// TIA Portal project "9input_to_4output" (V14)

(* hardware
DEVICE "S7-1200 station_1"  S7-1200 Station
   slot 0: "Rack_0"  S7-1200 Rack  Rack  V1.0
   slot 1: "PLC_1"  CPU 1214C DC/DC/DC  6ES7 214-1AG40-0XB0  V4.2
DEVICE "HMI_1"  KTP700 Basic PN
   slot 0: "KTP700 Basic PN"  KTP700 Basic PN  6AV2 123-2GB03-0AX0  14.0.1.0
   slot 1: "HMI_RT_1"  KTP700 Basic PN  6AV2 123-2GB03-0AX0  14.0.1.0
   slot 5: "HMI_1.IE_CP_1"  PROFINET Interface  14.0.1.0
      slot 1: "PROFINET Interface_1"  PROFINET Interface
         slot 1: "Port_1"  Port
*)

// ===== PLC "PLC_1"  CPU 1214C DC/DC/DC =====

VAR_GLOBAL   // PLC tag table "Default tag table"
   "nut1" AT %M0.0 : Bool;
   "nut3" AT %M0.1 : Bool;
   "nut4" AT %M0.2 : Bool;
   "nut7" AT %M0.3 : Bool;
   "nut2" AT %M0.5 : Bool;
   "nut6" AT %M0.6 : Bool;
   "Tag_7" AT %Q0.0 : Bool;
   "Tag_8" AT %Q0.1 : Bool;
   "nut5" AT %M0.7 : Bool;
   "nut9" AT %M0.4 : Bool;
   "nut8" AT %M1.0 : Bool;
   "den1" AT %Q0.4 : Bool;
   "den2" AT %Q0.5 : Bool;
   "den3" AT %Q0.6 : Bool;
   "den4" AT %Q0.7 : Bool;
END_VAR

ORGANIZATION_BLOCK "Main"   // OB1, LAD, ProgramCycle
TITLE = "Main Program Sweep (Cycle)"
{ S7_Optimized_Access := 'TRUE' }
VERSION : 0.1
   VAR_INPUT
      Initial_Call : Bool;   // Initial call of this OB
      Remanence : Bool;   // =True, if remanent data are available
   END_VAR
BEGIN

REGION Network 1
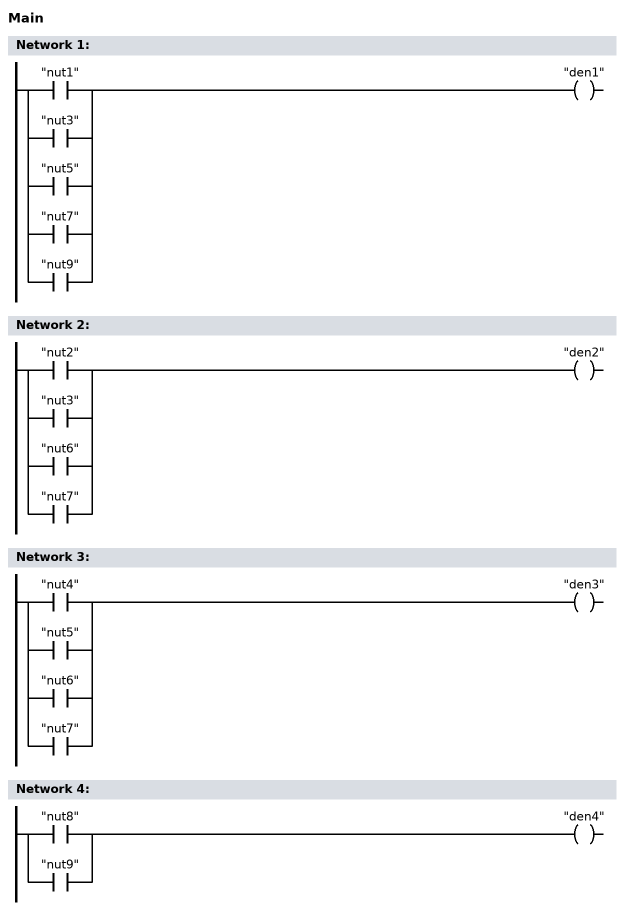
   RUNG wire#powerrail
      Contact( "nut1" )
      wire#w1
      Coil( "den1" )
   END_RUNG
   RUNG wire#powerrail
      Contact( "nut3" )
   END_RUNG wire#w1
   RUNG wire#powerrail
      Contact( "nut5" )
   END_RUNG wire#w1
   RUNG wire#powerrail
      Contact( "nut7" )
   END_RUNG wire#w1
   RUNG wire#powerrail
      Contact( "nut9" )
   END_RUNG wire#w1
   // the same network as SCL:
   "den1" := "nut1" OR "nut3" OR "nut5" OR "nut7" OR "nut9";
END_REGION

REGION Network 2
   RUNG wire#powerrail
      Contact( "nut2" )
      wire#w1
      Coil( "den2" )
   END_RUNG
   RUNG wire#powerrail
      Contact( "nut3" )
   END_RUNG wire#w1
   RUNG wire#powerrail
      Contact( "nut6" )
   END_RUNG wire#w1
   RUNG wire#powerrail
      Contact( "nut7" )
   END_RUNG wire#w1
   // the same network as SCL:
   "den2" := "nut2" OR "nut3" OR "nut6" OR "nut7";
END_REGION

REGION Network 3
   RUNG wire#powerrail
      Contact( "nut4" )
      wire#w1
      Coil( "den3" )
   END_RUNG
   RUNG wire#powerrail
      Contact( "nut5" )
   END_RUNG wire#w1
   RUNG wire#powerrail
      Contact( "nut6" )
   END_RUNG wire#w1
   RUNG wire#powerrail
      Contact( "nut7" )
   END_RUNG wire#w1
   // the same network as SCL:
   "den3" := "nut4" OR "nut5" OR "nut6" OR "nut7";
END_REGION

REGION Network 4
   RUNG wire#powerrail
      Contact( "nut8" )
      wire#w1
      Coil( "den4" )
   END_RUNG
   RUNG wire#powerrail
      Contact( "nut9" )
   END_RUNG wire#w1
   // the same network as SCL:
   "den4" := "nut8" OR "nut9";
END_REGION
END_ORGANIZATION_BLOCK

(* ===== HMI "HMI_RT_1" =====
system functions are stored by id; their names below are inferred from use
connection "HMI_Connection_1": ETHERNET, SMART_S7_1200_OMS

HMI tags "Default tag table"
   "Tag_ScreenNumber" : UInt, internal
   "nut1" : Bool = PLC nut1 AT %M0.0, 1 s
   "nut2" : Bool = PLC nut2 AT %M0.5, 1 s
   "nut3" : Bool = PLC nut3 AT %M0.1, 1 s
   "nut4" : Bool = PLC nut4 AT %M0.2, 1 s
   "nut5" : Bool = PLC nut5 AT %M0.7, 1 s
   "nut6" : Bool = PLC nut6 AT %M0.6, 1 s
   "nut7" : Bool = PLC nut7 AT %M0.3, 1 s
   "nut8" : Bool = PLC nut8 AT %M1.0, 1 s
   "nut9" : Bool = PLC nut9 AT %M0.4, 1 s
   "den1" : Bool = PLC den1 AT %Q0.4, 1 s
   "den2" : Bool = PLC den2 AT %Q0.5, 1 s
   "den3" : Bool = PLC den3 AT %Q0.6, 1 s
   "den4" : Bool = PLC den4 AT %Q0.7, 1 s

Template "Template_1" 800x480
   Button "Exit" at 714,429 size 71x50; TextOff 'Exit'; PictureOff "ExitRuntime_KTP700_Basic_PN_TR"; PictureOn "ExitRuntime_KTP700_Basic_PN_TR"
      on Release: StopRuntime(0)
   Button "Template_Button" at 614,429 size 71x50; TextOff 'Text'
   Button "Template_Button_1" at 514,429 size 71x50; TextOff 'Text'
   Button "Template_Button_2" at 414,429 size 71x50; TextOff 'Text'
   Button "Template_Button_3" at 314,429 size 71x50; TextOff 'Text'
   Button "Template_Button_4" at 214,429 size 71x50; TextOff 'Text'
   Button "Alarms" at 114,429 size 71x50; TextOff 'Alarms'; PictureOff "AlarmDisplay_KTP700_Basic_PN_TR"; PictureOn "AlarmDisplay_KTP700_Basic_PN_TR"
      on Release: function_ef3f5d25("Alarm window_Unacknowledged", -1)
   Button "Start screen" at 14,429 size 71x50; TextOff 'Start screen'; PictureOff "NavigateHome_KTP700_Basic_PN_TR"; PictureOn "NavigateHome_KTP700_Basic_PN_TR"
      on Release: ActivateScreen("Root screen", 0)
   SymbolicIOField "Symbolic_IO_Field_Screen" at 93,9 size 600x33; TextOff '0'; TextOn '1'; TextList "TextList_ScreenNames"
      ProcessValue <- "Tag_ScreenNumber"
      on Change: ActivateScreenByNumber("Tag_ScreenNumber", 0)
   DateTimeField "HmiScreenItemData" at 695,25 size 105x25
   DateTimeField "HmiScreenItemData_1" at 695,0 size 105x25
   GraphicView "Logo" at 0,0 size 91x51; Picture "Logo of HMI_1"

screen "Root screen" 800x480, template "Template_1"
   on GenerateScreen: SetTag("Tag_ScreenNumber", 1)
   Circle "Circle_1" at 733,119 size 48x48
      Appearance <- "den1"
   Circle "Circle_2" at 666,119 size 48x48
      Appearance <- "den2"
   Circle "Circle_3" at 595,119 size 48x48
      Appearance <- "den3"
   Circle "Circle_4" at 514,119 size 48x48
      Appearance <- "den4"
   TextField "Text field_1" at 742,175 size 27x23; Text 'D1'
   TextField "Text field_2" at 678,174 size 27x23; Text 'D2'
   TextField "Text field_3" at 604,174 size 27x23; Text 'D3'
   TextField "Text field_4" at 527,173 size 27x23; Text 'D4'
   Switch "Switch_1" at 118,87 size 64x32; CaptionText 'Switch'; TextOff 'OFF'; TextOn 'ON'
      on SwitchOn: SetBit("nut1")
      on SwitchOff: ResetBit("nut1")
   TextField "Text field_5" at 142,124 size 15x23; Text '1'
   Switch "Switch_2" at 215,89 size 64x32; TextOn 'ON'; CaptionText 'Switch'; TextOff 'OFF'
      on SwitchOff: ResetBit("nut2")
      on SwitchOn: SetBit("nut2")
   Switch "Switch_3" at 314,87 size 64x32; TextOn 'ON'; CaptionText 'Switch'; TextOff 'OFF'
      on SwitchOn: SetBit("nut3")
      on SwitchOff: ResetBit("nut3")
   Switch "Switch_4" at 414,89 size 64x32; TextOn 'ON'; CaptionText 'Switch'; TextOff 'OFF'
      on SwitchOff: ResetBit("nut4")
      on SwitchOn: SetBit("nut4")
   Switch "Switch_5" at 18,89 size 64x32; TextOn 'ON'; CaptionText 'Switch'; TextOff 'OFF'
   TextField "Text field_6" at 45,123 size 15x23; Text '0'
   TextField "Text field_7" at 246,123 size 15x23; Text '2'
   TextField "Text field_8" at 343,123 size 15x23; Text '3'
   TextField "Text field_9" at 442,123 size 15x23; Text '4'
   Switch "Switch_6" at 118,165 size 64x32; TextOn 'ON'; CaptionText 'Switch'; TextOff 'OFF'
      on SwitchOff: ResetBit("nut6")
      on SwitchOn: SetBit("nut6")
   TextField "Text field_10" at 142,202 size 15x23; Text '6'
   Switch "Switch_7" at 215,167 size 64x32; TextOn 'ON'; CaptionText 'Switch'; TextOff 'OFF'
      on SwitchOn: SetBit("nut7")
      on SwitchOff: ResetBit("nut7")
   Switch "Switch_8" at 314,165 size 64x32; TextOn 'ON'; CaptionText 'Switch'; TextOff 'OFF'
      on SwitchOff: ResetBit("nut8")
      on SwitchOn: SetBit("nut8")
   Switch "Switch_9" at 414,167 size 64x32; TextOn 'ON'; CaptionText 'Switch'; TextOff 'OFF'
      on SwitchOn: SetBit("nut9")
      on SwitchOff: ResetBit("nut9")
   Switch "Switch_10" at 18,167 size 64x32; TextOn 'ON'; CaptionText 'Switch'; TextOff 'OFF'
      on SwitchOn: SetBit("nut5")
      on SwitchOff: ResetBit("nut5")
   TextField "Text field_11" at 45,201 size 15x23; Text '5'
   TextField "Text field_12" at 246,201 size 15x23; Text '7'
   TextField "Text field_13" at 343,201 size 15x23; Text '8'
   TextField "Text field_14" at 442,201 size 15x23; Text '9'
*)